// TIA Portal V19 export
FUNCTION_BLOCK "Ventil_Stati"   // FB1095, LAD
TITLE = Ventilstatus
{ S7_Optimized_Access := 'TRUE' }
// 0: geschlossen (grau)
// 1: geöffnet (grün)
// 2: Störung (rot)
// stored: AutoNumber false, MemoryReserve 100, SetENOAutomatically false
   VAR RETAIN
      Param { ExternalAccessible := 'False'; ExternalVisible := 'False'; ExternalWritable := 'False'} : Struct
         "TO" : Time := T#20s;
      END_STRUCT;
      Mld : Struct
         "TO_auf_CM01.QM18" : Bool;
         "TO_zu_CM01.QM18" : Bool;
         "SF_CM01.QM18" : Bool;
         "TO_auf_CM01.QM19" : Bool;
         "TO_zu_CM01.QM19" : Bool;
         "SF_CM01.QM19" : Bool;
         "TO_auf_CM01.QM20" : Bool;
         "TO_zu_CM01.QM20" : Bool;
         "SF_CM01.QM20" : Bool;
         "TO_auf_CM01.QM25" : Bool;
         "TO_zu_CM01.QM25" : Bool;
         "SF_CM01.QM25" : Bool;
         "TO_auf_CM01.QM26" : Bool;
         "TO_zu_CM01.QM26" : Bool;
         "SF_CM01.QM26" : Bool;
         "TO_auf_CM01.QM27" : Bool;
         "TO_zu_CM01.QM27" : Bool;
         "SF_CM01.QM27" : Bool;
         "TO_auf_CM02.QM55" : Bool;
         "TO_zu_CM02.QM55" : Bool;
         "SF_CM02.QM55" : Bool;
         "TO_auf_CM02.QM56" : Bool;
         "TO_zu_CM02.QM56" : Bool;
         "SF_CM02.QM56" : Bool;
         "TO_auf_CM02.QM57" : Bool;
         "TO_zu_CM02.QM57" : Bool;
         "SF_CM02.QM57" : Bool;
         "TO_auf_CM02.QM62" : Bool;
         "TO_zu_CM02.QM62" : Bool;
         "SF_CM02.QM62" : Bool;
         "TO_auf_CM02.QM63" : Bool;
         "TO_zu_CM02.QM63" : Bool;
         "SF_CM02.QM63" : Bool;
         "TO_auf_CM02.QM64" : Bool;
         "TO_zu_CM02.QM64" : Bool;
         "SF_CM02.QM64" : Bool;
         "TO_auf_HQ01.QM21" : Bool;
         "TO_zu_HQ01.QM21" : Bool;
         "SF_HQ01.QM21" : Bool;
         "TO_auf_HQ01.QM22" : Bool;
         "TO_zu_HQ01.QM22" : Bool;
         "SF_HQ01.QM22" : Bool;
         "TO_auf_HQ01.QM23" : Bool;
         "TO_zu_HQ01.QM23" : Bool;
         "SF_HQ01.QM23" : Bool;
         "TO_auf_HQ01.QM24" : Bool;
         "TO_zu_HQ01.QM24" : Bool;
         "SF_HQ01.QM24" : Bool;
         "TO_auf_HQ01.LV01" : Bool;
         "TO_zu_HQ01.LV01" : Bool;
         "SF_HQ01.LV01" : Bool;
         "TO_auf_HQ02.QM58" : Bool;
         "TO_zu_HQ02.QM58" : Bool;
         "SF_HQ02.QM58" : Bool;
         "TO_auf_HQ02.QM59" : Bool;
         "TO_zu_HQ02.QM59" : Bool;
         "SF_HQ02.QM59" : Bool;
         "TO_auf_HQ02.QM60" : Bool;
         "TO_zu_HQ02.QM60" : Bool;
         "SF_HQ02.QM60" : Bool;
         "TO_auf_HQ02.QM61" : Bool;
         "TO_zu_HQ02.QM61" : Bool;
         "SF_HQ02.QM61" : Bool;
         "TO_auf_HQ02.LV02" : Bool;
         "TO_zu_HQ02.LV02" : Bool;
         "SF_HQ02.LV02" : Bool;
         "TO_auf_CM03.QM33" : Bool;
         "TO_zu_CM03.QM33" : Bool;
         "SF_CM03.QM33" : Bool;
         "TO_auf_CM03.QM34" : Bool;
         "TO_zu_CM03.QM34" : Bool;
         "SF_CM03.QM34" : Bool;
         "TO_auf_CM04.QM72" : Bool;
         "TO_zu_CM04.QM72" : Bool;
         "SF_CM04.QM72" : Bool;
         "TO_auf_CM04.QM73" : Bool;
         "TO_zu_CM04.QM73" : Bool;
         "SF_CM04.QM73" : Bool;
         "TO_auf_CM05.QM61" : Bool;
         "TO_zu_CM05.QM61" : Bool;
         "SF_CM05.QM61" : Bool;
         "TO_auf_CM05.QM64" : Bool;
         "TO_zu_CM05.QM64" : Bool;
         "SF_CM05.QM64" : Bool;
         "TO_auf_GP01.QM14" : Bool;
         "TO_zu_GP01.QM14" : Bool;
         "SF_GP01.QM14" : Bool;
         "TO_auf_GP01.QM15" : Bool;
         "TO_zu_GP01.QM15" : Bool;
         "SF_GP01.QM15" : Bool;
         "TO_auf_GP01.QM16" : Bool;
         "TO_zu_GP01.QM16" : Bool;
         "SF_GP01.QM16" : Bool;
         "TO_auf_GP01.QM17" : Bool;
         "TO_zu_GP01.QM17" : Bool;
         "SF_GP01.QM17" : Bool;
         "TO_auf_GP01.QM18" : Bool;
         "TO_zu_GP01.QM18" : Bool;
         "SF_GP01.QM18" : Bool;
         "TO_auf_GP01.QM19" : Bool;
         "TO_zu_GP01.QM19" : Bool;
         "SF_GP01.QM19" : Bool;
         "TO_auf_GP01.QM20" : Bool;
         "TO_zu_GP01.QM20" : Bool;
         "SF_GP01.QM20" : Bool;
         "TO_auf_GP01.QM21" : Bool;
         "TO_zu_GP01.QM21" : Bool;
         "SF_GP01.QM21" : Bool;
         "TO_auf_GP01.QM22" : Bool;
         "TO_zu_GP01.QM22" : Bool;
         "SF_GP01.QM22" : Bool;
         "TO_auf_GP02.QM38" : Bool;
         "TO_zu_GP02.QM38" : Bool;
         "SF_GP02.QM38" : Bool;
         "TO_auf_GP02.QM39" : Bool;
         "TO_zu_GP02.QM39" : Bool;
         "SF_GP02.QM39" : Bool;
         "TO_auf_GP02.QM40" : Bool;
         "TO_zu_GP02.QM40" : Bool;
         "SF_GP02.QM40" : Bool;
         "TO_auf_GP02.QM41" : Bool;
         "TO_zu_GP02.QM41" : Bool;
         "SF_GP02.QM41" : Bool;
         "TO_auf_GP02.QM42" : Bool;
         "TO_zu_GP02.QM42" : Bool;
         "SF_GP02.QM42" : Bool;
         "TO_auf_GP02.QM43" : Bool;
         "TO_zu_GP02.QM43" : Bool;
         "SF_GP02.QM43" : Bool;
         "TO_auf_GP02.QM44" : Bool;
         "TO_zu_GP02.QM44" : Bool;
         "SF_GP02.QM44" : Bool;
         "TO_auf_GP02.QM45" : Bool;
         "TO_zu_GP02.QM45" : Bool;
         "SF_GP02.QM45" : Bool;
         "TO_auf_GP02.QM46" : Bool;
         "TO_zu_GP02.QM46" : Bool;
         "SF_GP02.QM46" : Bool;
      END_STRUCT;
   END_VAR
   VAR
      IEC_Timer { ExternalAccessible := 'False'; ExternalVisible := 'False'; ExternalWritable := 'False'} : Struct
         "TO_auf_CM01.QM18" { S7_SetPoint := 'True'} : TON_TIME;
         "TO_zu_CM01.QM18" { S7_SetPoint := 'True'} : TON_TIME;
         "TO_auf_CM01.QM19" { S7_SetPoint := 'True'} : TON_TIME;
         "TO_zu_CM01.QM19" { S7_SetPoint := 'True'} : TON_TIME;
         "TO_auf_CM01.QM20" { S7_SetPoint := 'True'} : TON_TIME;
         "TO_zu_CM01.QM20" { S7_SetPoint := 'True'} : TON_TIME;
         "TO_auf_CM01.QM25" { S7_SetPoint := 'True'} : TON_TIME;
         "TO_zu_CM01.QM25" { S7_SetPoint := 'True'} : TON_TIME;
         "TO_auf_CM01.QM26" { S7_SetPoint := 'True'} : TON_TIME;
         "TO_zu_CM01.QM26" { S7_SetPoint := 'True'} : TON_TIME;
         "TO_auf_CM01.QM27" { S7_SetPoint := 'True'} : TON_TIME;
         "TO_zu_CM01.QM27" { S7_SetPoint := 'True'} : TON_TIME;
         "TO_auf_CM02.QM55" { S7_SetPoint := 'True'} : TON_TIME;
         "TO_zu_CM02.QM55" { S7_SetPoint := 'True'} : TON_TIME;
         "TO_auf_CM02.QM56" { S7_SetPoint := 'True'} : TON_TIME;
         "TO_zu_CM02.QM56" { S7_SetPoint := 'True'} : TON_TIME;
         "TO_auf_CM02.QM57" { S7_SetPoint := 'True'} : TON_TIME;
         "TO_zu_CM02.QM57" { S7_SetPoint := 'True'} : TON_TIME;
         "TO_auf_CM02.QM62" { S7_SetPoint := 'True'} : TON_TIME;
         "TO_zu_CM02.QM62" { S7_SetPoint := 'True'} : TON_TIME;
         "TO_auf_CM02.QM63" { S7_SetPoint := 'True'} : TON_TIME;
         "TO_zu_CM02.QM63" { S7_SetPoint := 'True'} : TON_TIME;
         "TO_auf_CM02.QM64" { S7_SetPoint := 'True'} : TON_TIME;
         "TO_zu_CM02.QM64" { S7_SetPoint := 'True'} : TON_TIME;
         "TO_auf_HQ01.QM21" { S7_SetPoint := 'True'} : TON_TIME;
         "TO_zu_HQ01.QM21" { S7_SetPoint := 'True'} : TON_TIME;
         "TO_auf_HQ01.QM22" { S7_SetPoint := 'True'} : TON_TIME;
         "TO_zu_HQ01.QM22" { S7_SetPoint := 'True'} : TON_TIME;
         "TO_auf_HQ01.QM23" { S7_SetPoint := 'True'} : TON_TIME;
         "TO_zu_HQ01.QM23" { S7_SetPoint := 'True'} : TON_TIME;
         "TO_auf_HQ01.QM24" { S7_SetPoint := 'True'} : TON_TIME;
         "TO_zu_HQ01.QM24" { S7_SetPoint := 'True'} : TON_TIME;
         "TO_auf_HQ01.LV01" { S7_SetPoint := 'True'} : TON_TIME;
         "TO_zu_HQ01.LV01" { S7_SetPoint := 'True'} : TON_TIME;
         "TO_auf_HQ02.QM58" { S7_SetPoint := 'True'} : TON_TIME;
         "TO_zu_HQ02.QM58" { S7_SetPoint := 'True'} : TON_TIME;
         "TO_auf_HQ02.QM59" { S7_SetPoint := 'True'} : TON_TIME;
         "TO_zu_HQ02.QM59" { S7_SetPoint := 'True'} : TON_TIME;
         "TO_auf_HQ02.QM60" { S7_SetPoint := 'True'} : TON_TIME;
         "TO_zu_HQ02.QM60" { S7_SetPoint := 'True'} : TON_TIME;
         "TO_auf_HQ02.QM61" { S7_SetPoint := 'True'} : TON_TIME;
         "TO_zu_HQ02.QM61" { S7_SetPoint := 'True'} : TON_TIME;
         "TO_auf_HQ02.LV02" { S7_SetPoint := 'True'} : TON_TIME;
         "TO_zu_HQ02.LV02" { S7_SetPoint := 'True'} : TON_TIME;
         "TO_auf_CM03.QM33" { S7_SetPoint := 'True'} : TON_TIME;
         "TO_zu_CM03.QM33" { S7_SetPoint := 'True'} : TON_TIME;
         "TO_auf_CM03.QM34" { S7_SetPoint := 'True'} : TON_TIME;
         "TO_zu_CM03.QM34" { S7_SetPoint := 'True'} : TON_TIME;
         "TO_auf_CM04.QM72" { S7_SetPoint := 'True'} : TON_TIME;
         "TO_zu_CM04.QM72" { S7_SetPoint := 'True'} : TON_TIME;
         "TO_auf_CM04.QM73" { S7_SetPoint := 'True'} : TON_TIME;
         "TO_zu_CM04.QM73" { S7_SetPoint := 'True'} : TON_TIME;
         "TO_auf_CM05.QM61" { S7_SetPoint := 'True'} : TON_TIME;
         "TO_zu_CM05.QM61" { S7_SetPoint := 'True'} : TON_TIME;
         "TO_auf_CM05.QM64" { S7_SetPoint := 'True'} : TON_TIME;
         "TO_zu_CM05.QM64" { S7_SetPoint := 'True'} : TON_TIME;
         "TO_auf_GP01.QM14" { S7_SetPoint := 'True'} : TON_TIME;
         "TO_zu_GP01.QM14" { S7_SetPoint := 'True'} : TON_TIME;
         "TO_auf_GP01.QM15" { S7_SetPoint := 'True'} : TON_TIME;
         "TO_zu_GP01.QM15" { S7_SetPoint := 'True'} : TON_TIME;
         "TO_auf_GP01.QM16" { S7_SetPoint := 'True'} : TON_TIME;
         "TO_zu_GP01.QM16" { S7_SetPoint := 'True'} : TON_TIME;
         "TO_auf_GP01.QM17" { S7_SetPoint := 'True'} : TON_TIME;
         "TO_zu_GP01.QM17" { S7_SetPoint := 'True'} : TON_TIME;
         "TO_auf_GP01.QM18" { S7_SetPoint := 'True'} : TON_TIME;
         "TO_zu_GP01.QM18" { S7_SetPoint := 'True'} : TON_TIME;
         "TO_auf_GP01.QM19" { S7_SetPoint := 'True'} : TON_TIME;
         "TO_zu_GP01.QM19" { S7_SetPoint := 'True'} : TON_TIME;
         "TO_auf_GP01.QM20" { S7_SetPoint := 'True'} : TON_TIME;
         "TO_zu_GP01.QM20" { S7_SetPoint := 'True'} : TON_TIME;
         "TO_auf_GP01.QM21" { S7_SetPoint := 'True'} : TON_TIME;
         "TO_zu_GP01.QM21" { S7_SetPoint := 'True'} : TON_TIME;
         "TO_auf_GP01.QM22" { S7_SetPoint := 'True'} : TON_TIME;
         "TO_zu_GP01.QM22" { S7_SetPoint := 'True'} : TON_TIME;
         "TO_auf_GP02.QM38" { S7_SetPoint := 'True'} : TON_TIME;
         "TO_zu_GP02.QM38" { S7_SetPoint := 'True'} : TON_TIME;
         "TO_auf_GP02.QM39" { S7_SetPoint := 'True'} : TON_TIME;
         "TO_zu_GP02.QM39" { S7_SetPoint := 'True'} : TON_TIME;
         "TO_auf_GP02.QM40" { S7_SetPoint := 'True'} : TON_TIME;
         "TO_zu_GP02.QM40" { S7_SetPoint := 'True'} : TON_TIME;
         "TO_auf_GP02.QM41" { S7_SetPoint := 'True'} : TON_TIME;
         "TO_zu_GP02.QM41" { S7_SetPoint := 'True'} : TON_TIME;
         "TO_auf_GP02.QM42" { S7_SetPoint := 'True'} : TON_TIME;
         "TO_zu_GP02.QM42" { S7_SetPoint := 'True'} : TON_TIME;
         "TO_auf_GP02.QM43" { S7_SetPoint := 'True'} : TON_TIME;
         "TO_zu_GP02.QM43" { S7_SetPoint := 'True'} : TON_TIME;
         "TO_auf_GP02.QM44" { S7_SetPoint := 'True'} : TON_TIME;
         "TO_zu_GP02.QM44" { S7_SetPoint := 'True'} : TON_TIME;
         "TO_auf_GP02.QM45" { S7_SetPoint := 'True'} : TON_TIME;
         "TO_zu_GP02.QM45" { S7_SetPoint := 'True'} : TON_TIME;
         "TO_auf_GP02.QM46" { S7_SetPoint := 'True'} : TON_TIME;
         "TO_zu_GP02.QM46" { S7_SetPoint := 'True'} : TON_TIME;
      END_STRUCT;
   END_VAR
   VAR CONSTANT
      grau : USInt;
      grün : USInt := 1;
      rot : USInt := 2;
   END_VAR
BEGIN

REGION Network 1 (SCL): CM01

   "Ventilstatus"(SRM_auf:= "E_SRM_CM01.QM18_auf",
                  SRM_zu:= "E_SRM_CM01.QM18_zu",
                  A_Ventil:= "A_CM01.QM18",
                  Zeit:= #Param.TO,
                  "Farbe HMI"=> "Panel".Ventil."CM01.QM18",
                  Mld_Sensorfehler:= #Mld."SF_CM01.QM18",
                  Mld_TO_oeffnen=> #Mld."TO_auf_CM01.QM18",
                  Mld_TO_schliessen=> #Mld."TO_zu_CM01.QM18",
                  TO_oeffnen:= #IEC_Timer."TO_auf_CM01.QM18",
                  TO_schliessen:= #IEC_Timer."TO_zu_CM01.QM18");

   "Ventilstatus"(SRM_auf := "E_SRM_CM01.QM19_auf",
                  SRM_zu := "E_SRM_CM01.QM19_zu",
                  A_Ventil := "A_CM01.QM19",
                  Zeit := #Param.TO,
                  "Farbe HMI" => "Panel".Ventil."CM01.QM19",
                  Mld_Sensorfehler := #Mld."SF_CM01.QM19",
                  Mld_TO_oeffnen => #Mld."TO_auf_CM01.QM19",
                  Mld_TO_schliessen => #Mld."TO_zu_CM01.QM19",
                  TO_oeffnen := #IEC_Timer."TO_auf_CM01.QM19",
                  TO_schliessen := #IEC_Timer."TO_zu_CM01.QM19");

   "Ventilstatus"(SRM_auf := "E_SRM_CM01.QM20_auf",
                  SRM_zu := "E_SRM_CM01.QM20_zu",
                  A_Ventil := "A_CM01.QM20",
                  Zeit := #Param.TO,
                  "Farbe HMI" => "Panel".Ventil."CM01.QM20",
                  Mld_Sensorfehler := #Mld."SF_CM01.QM20",
                  Mld_TO_oeffnen => #Mld."TO_auf_CM01.QM20",
                  Mld_TO_schliessen => #Mld."TO_zu_CM01.QM20",
                  TO_oeffnen := #IEC_Timer."TO_auf_CM01.QM20",
                  TO_schliessen := #IEC_Timer."TO_zu_CM01.QM20");

   "Ventilstatus"(SRM_auf := "E_SRM_CM01.QM25_auf",
                  SRM_zu := "E_SRM_CM01.QM25_zu",
                  A_Ventil := "A_CM01.QM25",
                  Zeit := #Param.TO,
                  "Farbe HMI" => "Panel".Ventil."CM01.QM25",
                  Mld_Sensorfehler := #Mld."SF_CM01.QM25",
                  Mld_TO_oeffnen => #Mld."TO_auf_CM01.QM25",
                  Mld_TO_schliessen => #Mld."TO_zu_CM01.QM25",
                  TO_oeffnen := #IEC_Timer."TO_auf_CM01.QM25",
                  TO_schliessen := #IEC_Timer."TO_zu_CM01.QM25");

   "Ventilstatus"(SRM_auf := "E_SRM_CM01.QM26_auf",
                  SRM_zu := "E_SRM_CM01.QM26_zu",
                  A_Ventil := "A_CM01.QM26",
                  Zeit := #Param.TO,
                  "Farbe HMI" => "Panel".Ventil."CM01.QM26",
                  Mld_Sensorfehler := #Mld."SF_CM01.QM26",
                  Mld_TO_oeffnen => #Mld."TO_auf_CM01.QM26",
                  Mld_TO_schliessen => #Mld."TO_zu_CM01.QM26",
                  TO_oeffnen := #IEC_Timer."TO_auf_CM01.QM26",
                  TO_schliessen := #IEC_Timer."TO_zu_CM01.QM26");

   "Ventilstatus"(SRM_auf := "E_SRM_CM01.QM27_auf",
                  SRM_zu := "E_SRM_CM01.QM27_zu",
                  A_Ventil := "A_CM01.QM27",
                  Zeit := #Param.TO,
                  "Farbe HMI" => "Panel".Ventil."CM01.QM27",
                  Mld_Sensorfehler := #Mld."SF_CM01.QM27",
                  Mld_TO_oeffnen => #Mld."TO_auf_CM01.QM27",
                  Mld_TO_schliessen => #Mld."TO_zu_CM01.QM27",
                  TO_oeffnen := #IEC_Timer."TO_auf_CM01.QM27",
                  TO_schliessen := #IEC_Timer."TO_zu_CM01.QM27");
END_REGION

REGION Network 2 (SCL): HQ01
   "Ventilstatus"(SRM_auf := "E_SRM_HQ01.LV01_auf",
                  SRM_zu := "E_SRM_HQ01.LV01_zu",
                  A_Ventil := "A_HQ01.LV01",
                  Zeit := #Param.TO,
                  "Farbe HMI" => "Panel".Ventil."HQ01.LV01",
                  Mld_Sensorfehler := #Mld."SF_HQ01.LV01",
                  Mld_TO_oeffnen => #Mld."TO_auf_HQ01.LV01",
                  Mld_TO_schliessen => #Mld."TO_zu_HQ01.LV01",
                  TO_oeffnen := #IEC_Timer."TO_auf_HQ01.LV01",
                  TO_schliessen := #IEC_Timer."TO_zu_HQ01.LV01");

   "Ventilstatus"(SRM_auf := "E_SRM_HQ01.QM21_auf",
                  SRM_zu := "E_SRM_HQ01.QM21_zu",
                  A_Ventil := "A_HQ01.QM21",
                  Zeit := #Param.TO,
                  "Farbe HMI" => "Panel".Ventil."HQ01.QM21",
                  Mld_Sensorfehler := #Mld."SF_HQ01.QM21",
                  Mld_TO_oeffnen => #Mld."TO_auf_HQ01.QM21",
                  Mld_TO_schliessen => #Mld."TO_zu_HQ01.QM21",
                  TO_oeffnen := #IEC_Timer."TO_auf_HQ01.QM21",
                  TO_schliessen := #IEC_Timer."TO_zu_HQ01.QM21");

   "Ventilstatus"(SRM_auf := "E_SRM_HQ01.QM22_auf",
                  SRM_zu := "E_SRM_HQ01.QM22_zu",
                  A_Ventil := "A_HQ01.QM22",
                  Zeit := #Param.TO,
                  "Farbe HMI" => "Panel".Ventil."HQ01.QM22",
                  Mld_Sensorfehler := #Mld."SF_HQ01.QM22",
                  Mld_TO_oeffnen => #Mld."TO_auf_HQ01.QM22",
                  Mld_TO_schliessen => #Mld."TO_zu_HQ01.QM22",
                  TO_oeffnen := #IEC_Timer."TO_auf_HQ01.QM22",
                  TO_schliessen := #IEC_Timer."TO_zu_HQ01.QM22");

   "Ventilstatus"(SRM_auf := "E_SRM_HQ01.QM23_auf",
                  SRM_zu := "E_SRM_HQ01.QM23_zu",
                  A_Ventil := "A_HQ01.QM23",
                  Zeit := #Param.TO,
                  "Farbe HMI" => "Panel".Ventil."HQ01.QM23",
                  Mld_Sensorfehler := #Mld."SF_HQ01.QM23",
                  Mld_TO_oeffnen => #Mld."TO_auf_HQ01.QM23",
                  Mld_TO_schliessen => #Mld."TO_zu_HQ01.QM23",
                  TO_oeffnen := #IEC_Timer."TO_auf_HQ01.QM23",
                  TO_schliessen := #IEC_Timer."TO_zu_HQ01.QM23");

   "Ventilstatus"(SRM_auf := "E_SRM_HQ01.QM24_auf",
                  SRM_zu := "E_SRM_HQ01.QM24_zu",
                  A_Ventil := "A_HQ01.QM24",
                  Zeit := #Param.TO,
                  "Farbe HMI" => "Panel".Ventil."HQ01.QM24",
                  Mld_Sensorfehler := #Mld."SF_HQ01.QM24",
                  Mld_TO_oeffnen => #Mld."TO_auf_HQ01.QM24",
                  Mld_TO_schliessen => #Mld."TO_zu_HQ01.QM24",
                  TO_oeffnen := #IEC_Timer."TO_auf_HQ01.QM24",
                  TO_schliessen := #IEC_Timer."TO_zu_HQ01.QM24");
END_REGION

REGION Network 3 (SCL): CM03

   "Ventilstatus"(SRM_auf := "E_SRM_CM03.QM33_auf",
                  SRM_zu := "E_SRM_CM03.QM33_zu",
                  A_Ventil := "A_CM03.QM33",
                  Zeit := #Param.TO,
                  "Farbe HMI" => "Panel".Ventil."CM03.QM33",
                  Mld_Sensorfehler := #Mld."SF_CM03.QM33",
                  Mld_TO_oeffnen => #Mld."TO_auf_CM03.QM33",
                  Mld_TO_schliessen => #Mld."TO_zu_CM03.QM33",
                  TO_oeffnen := #IEC_Timer."TO_auf_CM03.QM33",
                  TO_schliessen := #IEC_Timer."TO_zu_CM03.QM33");

   "Ventilstatus"(SRM_auf := "E_SRM_CM03.QM34_auf",
                  SRM_zu := "E_SRM_CM03.QM34_zu",
                  A_Ventil := "A_CM03.QM34",
                  Zeit := #Param.TO,
                  "Farbe HMI" => "Panel".Ventil."CM03.QM34",
                  Mld_Sensorfehler := #Mld."SF_CM03.QM34",
                  Mld_TO_oeffnen => #Mld."TO_auf_CM03.QM34",
                  Mld_TO_schliessen => #Mld."TO_zu_CM03.QM34",
                  TO_oeffnen := #IEC_Timer."TO_auf_CM03.QM34",
                  TO_schliessen := #IEC_Timer."TO_zu_CM03.QM34");

   "Ventilstatus_einfach"(A_Ventil:="A_CM03.QM35",
                          "Farbe HMI"=>"Panel".Ventil."CM03.QM35");

   "Ventilstatus_einfach"(A_Ventil := "A_CM03.QM36",
                          "Farbe HMI" => "Panel".Ventil."CM03.QM36");

   "Ventilstatus_einfach"(A_Ventil := "A_CM03.QM37",
                          "Farbe HMI" => "Panel".Ventil."CM03.QM37");
END_REGION

REGION Network 4 (SCL): CM02

   "Ventilstatus"(SRM_auf := "E_SRM_CM02.QM55_auf",
                  SRM_zu := "E_SRM_CM02.QM55_zu",
                  A_Ventil := "A_CM02.QM55",
                  Zeit := #Param.TO,
                  "Farbe HMI" => "Panel".Ventil."CM02.QM55",
                  Mld_Sensorfehler := #Mld."SF_CM02.QM55",
                  Mld_TO_oeffnen => #Mld."TO_auf_CM02.QM55",
                  Mld_TO_schliessen => #Mld."TO_zu_CM02.QM55",
                  TO_oeffnen := #IEC_Timer."TO_auf_CM02.QM55",
                  TO_schliessen := #IEC_Timer."TO_zu_CM02.QM55");

   "Ventilstatus"(SRM_auf := "E_SRM_CM02.QM56_auf",
                  SRM_zu := "E_SRM_CM02.QM56_zu",
                  A_Ventil := "A_CM02.QM56",
                  Zeit := #Param.TO,
                  "Farbe HMI" => "Panel".Ventil."CM02.QM56",
                  Mld_Sensorfehler := #Mld."SF_CM02.QM56",
                  Mld_TO_oeffnen => #Mld."TO_auf_CM02.QM56",
                  Mld_TO_schliessen => #Mld."TO_zu_CM02.QM56",
                  TO_oeffnen := #IEC_Timer."TO_auf_CM02.QM56",
                  TO_schliessen := #IEC_Timer."TO_zu_CM02.QM56");

   "Ventilstatus"(SRM_auf := "E_SRM_CM02.QM57_auf",
                  SRM_zu := "E_SRM_CM02.QM57_zu",
                  A_Ventil := "A_CM02.QM57",
                  Zeit := #Param.TO,
                  "Farbe HMI" => "Panel".Ventil."CM02.QM57",
                  Mld_Sensorfehler := #Mld."SF_CM02.QM57",
                  Mld_TO_oeffnen => #Mld."TO_auf_CM02.QM57",
                  Mld_TO_schliessen => #Mld."TO_zu_CM02.QM57",
                  TO_oeffnen := #IEC_Timer."TO_auf_CM02.QM57",
                  TO_schliessen := #IEC_Timer."TO_zu_CM02.QM57");

   "Ventilstatus"(SRM_auf := "E_SRM_CM02.QM62_auf",
                  SRM_zu := "E_SRM_CM02.QM62_zu",
                  A_Ventil := "A_CM02.QM62",
                  Zeit := #Param.TO,
                  "Farbe HMI" => "Panel".Ventil."CM02.QM62",
                  Mld_Sensorfehler := #Mld."SF_CM02.QM62",
                  Mld_TO_oeffnen => #Mld."TO_auf_CM02.QM62",
                  Mld_TO_schliessen => #Mld."TO_zu_CM02.QM62",
                  TO_oeffnen := #IEC_Timer."TO_auf_CM02.QM62",
                  TO_schliessen := #IEC_Timer."TO_zu_CM02.QM62");

   "Ventilstatus"(SRM_auf := "E_SRM_CM02.QM63_auf",
                  SRM_zu := "E_SRM_CM02.QM63_zu",
                  A_Ventil := "A_CM02.QM63",
                  Zeit := #Param.TO,
                  "Farbe HMI" => "Panel".Ventil."CM02.QM63",
                  Mld_Sensorfehler := #Mld."SF_CM02.QM63",
                  Mld_TO_oeffnen => #Mld."TO_auf_CM02.QM63",
                  Mld_TO_schliessen => #Mld."TO_zu_CM02.QM63",
                  TO_oeffnen := #IEC_Timer."TO_auf_CM02.QM63",
                  TO_schliessen := #IEC_Timer."TO_zu_CM02.QM63");

   "Ventilstatus"(SRM_auf := "E_SRM_CM02.QM64_auf",
                  SRM_zu := "E_SRM_CM02.QM64_zu",
                  A_Ventil := "A_CM02.QM64",
                  Zeit := #Param.TO,
                  "Farbe HMI" => "Panel".Ventil."CM02.QM64",
                  Mld_Sensorfehler := #Mld."SF_CM02.QM64",
                  Mld_TO_oeffnen => #Mld."TO_auf_CM02.QM64",
                  Mld_TO_schliessen => #Mld."TO_zu_CM02.QM64",
                  TO_oeffnen := #IEC_Timer."TO_auf_CM02.QM64",
                  TO_schliessen := #IEC_Timer."TO_zu_CM02.QM64");
END_REGION

REGION Network 5 (SCL): HQ02
   "Ventilstatus"(SRM_auf := "E_SRM_HQ02.LV02_auf",
                  SRM_zu := "E_SRM_HQ02.LV02_zu",
                  A_Ventil := "A_HQ02.LV02",
                  Zeit := #Param.TO,
                  "Farbe HMI" => "Panel".Ventil."HQ02.LV02",
                  Mld_Sensorfehler := #Mld."SF_HQ02.LV02",
                  Mld_TO_oeffnen => #Mld."TO_auf_HQ02.LV02",
                  Mld_TO_schliessen => #Mld."TO_zu_HQ02.LV02",
                  TO_oeffnen := #IEC_Timer."TO_auf_HQ02.LV02",
                  TO_schliessen := #IEC_Timer."TO_zu_HQ02.LV02");

   "Ventilstatus"(SRM_auf := "E_SRM_HQ02.QM58_auf",
                  SRM_zu := "E_SRM_HQ02.QM58_zu",
                  A_Ventil := "A_HQ02.QM58",
                  Zeit := #Param.TO,
                  "Farbe HMI" => "Panel".Ventil."HQ02.QM58",
                  Mld_Sensorfehler := #Mld."SF_HQ02.QM58",
                  Mld_TO_oeffnen => #Mld."TO_auf_HQ02.QM58",
                  Mld_TO_schliessen => #Mld."TO_zu_HQ02.QM58",
                  TO_oeffnen := #IEC_Timer."TO_auf_HQ02.QM58",
                  TO_schliessen := #IEC_Timer."TO_zu_HQ02.QM58");

   "Ventilstatus"(SRM_auf := "E_SRM_HQ02.QM59_auf",
                  SRM_zu := "E_SRM_HQ02.QM59_zu",
                  A_Ventil := "A_HQ02.QM59",
                  Zeit := #Param.TO,
                  "Farbe HMI" => "Panel".Ventil."HQ02.QM59",
                  Mld_Sensorfehler := #Mld."SF_HQ02.QM59",
                  Mld_TO_oeffnen => #Mld."TO_auf_HQ02.QM59",
                  Mld_TO_schliessen => #Mld."TO_zu_HQ02.QM59",
                  TO_oeffnen := #IEC_Timer."TO_auf_HQ02.QM59",
                  TO_schliessen := #IEC_Timer."TO_zu_HQ02.QM59");

   "Ventilstatus"(SRM_auf := "E_SRM_HQ02.QM60_auf",
                  SRM_zu := "E_SRM_HQ02.QM60_zu",
                  A_Ventil := "A_HQ02.QM60",
                  Zeit := #Param.TO,
                  "Farbe HMI" => "Panel".Ventil."HQ02.QM60",
                  Mld_Sensorfehler := #Mld."SF_HQ02.QM60",
                  Mld_TO_oeffnen => #Mld."TO_auf_HQ02.QM60",
                  Mld_TO_schliessen => #Mld."TO_zu_HQ02.QM60",
                  TO_oeffnen := #IEC_Timer."TO_auf_HQ02.QM60",
                  TO_schliessen := #IEC_Timer."TO_zu_HQ02.QM60");

   "Ventilstatus"(SRM_auf := "E_SRM_HQ02.QM61_auf",
                  SRM_zu := "E_SRM_HQ02.QM61_zu",
                  A_Ventil := "A_HQ02.QM61",
                  Zeit := #Param.TO,
                  "Farbe HMI" => "Panel".Ventil."HQ02.QM61",
                  Mld_Sensorfehler := #Mld."SF_HQ02.QM61",
                  Mld_TO_oeffnen => #Mld."TO_auf_HQ02.QM61",
                  Mld_TO_schliessen => #Mld."TO_zu_HQ02.QM61",
                  TO_oeffnen := #IEC_Timer."TO_auf_HQ02.QM61",
                  TO_schliessen := #IEC_Timer."TO_zu_HQ02.QM61");
END_REGION

REGION Network 6 (SCL): CM04

   "Ventilstatus"(SRM_auf := "E_SRM_CM04.QM72_auf",
                  SRM_zu := "E_SRM_CM04.QM72_zu",
                  A_Ventil := "A_CM04.QM72",
                  Zeit := #Param.TO,
                  "Farbe HMI" => "Panel".Ventil."CM04.QM72",
                  Mld_Sensorfehler := #Mld."SF_CM04.QM72",
                  Mld_TO_oeffnen => #Mld."TO_auf_CM04.QM72",
                  Mld_TO_schliessen => #Mld."TO_zu_CM04.QM72",
                  TO_oeffnen := #IEC_Timer."TO_auf_CM04.QM72",
                  TO_schliessen := #IEC_Timer."TO_zu_CM04.QM72");

   "Ventilstatus"(SRM_auf := "E_SRM_CM04.QM73_auf",
                  SRM_zu := "E_SRM_CM04.QM73_zu",
                  A_Ventil := "A_CM04.QM73",
                  Zeit := #Param.TO,
                  "Farbe HMI" => "Panel".Ventil."CM04.QM73",
                  Mld_Sensorfehler := #Mld."SF_CM04.QM73",
                  Mld_TO_oeffnen => #Mld."TO_auf_CM04.QM73",
                  Mld_TO_schliessen => #Mld."TO_zu_CM04.QM73",
                  TO_oeffnen := #IEC_Timer."TO_auf_CM04.QM73",
                  TO_schliessen := #IEC_Timer."TO_zu_CM04.QM73");

   "Ventilstatus_einfach"(A_Ventil := "A_CM04.QM74",
                          "Farbe HMI" => "Panel".Ventil."CM04.QM74");

   "Ventilstatus_einfach"(A_Ventil := "A_CM04.QM75",
                          "Farbe HMI" => "Panel".Ventil."CM04.QM75");

   "Ventilstatus_einfach"(A_Ventil := "A_CM04.QM76",
                          "Farbe HMI" => "Panel".Ventil."CM04.QM76");

   "Ventilstatus_einfach"(A_Ventil := "A_CM04.QM77",
                          "Farbe HMI" => "Panel".Ventil."CM04.QM77");
END_REGION

REGION Network 7 (SCL): CM05
   "Ventilstatus"(SRM_auf := "E_SRM_CM05.QM61_auf",
                  SRM_zu := "E_SRM_CM05.QM61_zu",
                  A_Ventil := "A_CM05.QM61",
                  Zeit := #Param.TO,
                  "Farbe HMI" => "Panel".Ventil."CM05.QM61",
                  Mld_Sensorfehler := #Mld."SF_CM05.QM61",
                  Mld_TO_oeffnen => #Mld."TO_auf_CM05.QM61",
                  Mld_TO_schliessen => #Mld."TO_zu_CM05.QM61",
                  TO_oeffnen := #IEC_Timer."TO_auf_CM05.QM61",
                  TO_schliessen := #IEC_Timer."TO_zu_CM05.QM61");

   "Ventilstatus_einfach"(A_Ventil := "A_CM05.QM62",
                          "Farbe HMI" => "Panel".Ventil."CM05.QM62");

   "Ventilstatus_einfach"(A_Ventil := "A_CM05.QM63",
                          "Farbe HMI" => "Panel".Ventil."CM05.QM63");

   "Ventilstatus"(SRM_auf := "E_SRM_CM05.QM64_auf",
                  SRM_zu := "E_SRM_CM05.QM64_zu",
                  A_Ventil := "A_CM05.QM64",
                  Zeit := #Param.TO,
                  "Farbe HMI" => "Panel".Ventil."CM05.QM64",
                  Mld_Sensorfehler := #Mld."SF_CM05.QM64",
                  Mld_TO_oeffnen => #Mld."TO_auf_CM05.QM64",
                  Mld_TO_schliessen => #Mld."TO_zu_CM05.QM64",
                  TO_oeffnen := #IEC_Timer."TO_auf_CM05.QM64",
                  TO_schliessen := #IEC_Timer."TO_zu_CM05.QM64");
END_REGION

REGION Network 8 (SCL): GP01

   "Ventilstatus"(SRM_auf := "E_SRM_GP01.QM14_auf",
                  SRM_zu := "E_SRM_GP01.QM14_zu",
                  A_Ventil := "A_GP01.QM14",
                  Zeit := #Param.TO,
                  "Farbe HMI" => "Panel".Ventil."GP01.QM14",
                  Mld_Sensorfehler := #Mld."SF_GP01.QM14",
                  Mld_TO_oeffnen => #Mld."TO_auf_GP01.QM14",
                  Mld_TO_schliessen => #Mld."TO_zu_GP01.QM14",
                  TO_oeffnen := #IEC_Timer."TO_auf_GP01.QM14",
                  TO_schliessen := #IEC_Timer."TO_zu_GP01.QM14");

   "Ventilstatus"(SRM_auf := "E_SRM_GP01.QM15_auf",
                  SRM_zu := "E_SRM_GP01.QM15_zu",
                  A_Ventil := "A_GP01.QM15",
                  Zeit := #Param.TO,
                  "Farbe HMI" => "Panel".Ventil."GP01.QM15",
                  Mld_Sensorfehler := #Mld."SF_GP01.QM15",
                  Mld_TO_oeffnen => #Mld."TO_auf_GP01.QM15",
                  Mld_TO_schliessen => #Mld."TO_zu_GP01.QM15",
                  TO_oeffnen := #IEC_Timer."TO_auf_GP01.QM15",
                  TO_schliessen := #IEC_Timer."TO_zu_GP01.QM15");

   "Ventilstatus"(SRM_auf := "E_SRM_GP01.QM16_auf",
                  SRM_zu := "E_SRM_GP01.QM16_zu",
                  A_Ventil := "A_GP01.QM16",
                  Zeit := #Param.TO,
                  "Farbe HMI" => "Panel".Ventil."GP01.QM16",
                  Mld_Sensorfehler := #Mld."SF_GP01.QM16",
                  Mld_TO_oeffnen => #Mld."TO_auf_GP01.QM16",
                  Mld_TO_schliessen => #Mld."TO_zu_GP01.QM16",
                  TO_oeffnen := #IEC_Timer."TO_auf_GP01.QM16",
                  TO_schliessen := #IEC_Timer."TO_zu_GP01.QM16");

   "Ventilstatus"(SRM_auf := "E_SRM_GP01.QM17_auf",
                  SRM_zu := "E_SRM_GP01.QM17_zu",
                  A_Ventil := "A_GP01.QM17",
                  Zeit := #Param.TO,
                  "Farbe HMI" => "Panel".Ventil."GP01.QM17",
                  Mld_Sensorfehler := #Mld."SF_GP01.QM17",
                  Mld_TO_oeffnen => #Mld."TO_auf_GP01.QM17",
                  Mld_TO_schliessen => #Mld."TO_zu_GP01.QM17",
                  TO_oeffnen := #IEC_Timer."TO_auf_GP01.QM17",
                  TO_schliessen := #IEC_Timer."TO_zu_GP01.QM17");

   "Ventilstatus"(SRM_auf := "E_SRM_GP01.QM18_auf",
                  SRM_zu := "E_SRM_GP01.QM18_zu",
                  A_Ventil := "A_GP01.QM18",
                  Zeit := #Param.TO,
                  "Farbe HMI" => "Panel".Ventil."GP01.QM18",
                  Mld_Sensorfehler := #Mld."SF_GP01.QM18",
                  Mld_TO_oeffnen => #Mld."TO_auf_GP01.QM18",
                  Mld_TO_schliessen => #Mld."TO_zu_GP01.QM18",
                  TO_oeffnen := #IEC_Timer."TO_auf_GP01.QM18",
                  TO_schliessen := #IEC_Timer."TO_zu_GP01.QM18");

   "Ventilstatus"(SRM_auf := "E_SRM_GP01.QM19_auf",
                  SRM_zu := "E_SRM_GP01.QM19_zu",
                  A_Ventil := "A_GP01.QM19",
                  Zeit := #Param.TO,
                  "Farbe HMI" => "Panel".Ventil."GP01.QM19",
                  Mld_Sensorfehler := #Mld."SF_GP01.QM19",
                  Mld_TO_oeffnen => #Mld."TO_auf_GP01.QM19",
                  Mld_TO_schliessen => #Mld."TO_zu_GP01.QM19",
                  TO_oeffnen := #IEC_Timer."TO_auf_GP01.QM19",
                  TO_schliessen := #IEC_Timer."TO_zu_GP01.QM19");

   "Ventilstatus"(SRM_auf := "E_SRM_GP01.QM20_auf",
                  SRM_zu := "E_SRM_GP01.QM20_zu",
                  A_Ventil := "A_GP01.QM20",
                  Zeit := #Param.TO,
                  "Farbe HMI" => "Panel".Ventil."GP01.QM20",
                  Mld_Sensorfehler := #Mld."SF_GP01.QM20",
                  Mld_TO_oeffnen => #Mld."TO_auf_GP01.QM20",
                  Mld_TO_schliessen => #Mld."TO_zu_GP01.QM20",
                  TO_oeffnen := #IEC_Timer."TO_auf_GP01.QM20",
                  TO_schliessen := #IEC_Timer."TO_zu_GP01.QM20");

   "Ventilstatus"(SRM_auf := "E_SRM_GP01.QM21_auf",
                  SRM_zu := "E_SRM_GP01.QM21_zu",
                  A_Ventil := "A_GP01.QM21",
                  Zeit := #Param.TO,
                  "Farbe HMI" => "Panel".Ventil."GP01.QM21",
                  Mld_Sensorfehler := #Mld."SF_GP01.QM21",
                  Mld_TO_oeffnen => #Mld."TO_auf_GP01.QM21",
                  Mld_TO_schliessen => #Mld."TO_zu_GP01.QM21",
                  TO_oeffnen := #IEC_Timer."TO_auf_GP01.QM21",
                  TO_schliessen := #IEC_Timer."TO_zu_GP01.QM21");

   "Ventilstatus"(SRM_auf := "E_SRM_GP01.QM22_auf",
                  SRM_zu := "E_SRM_GP01.QM22_zu",
                  A_Ventil := "A_GP01.QM22",
                  Zeit := #Param.TO,
                  "Farbe HMI" => "Panel".Ventil."GP01.QM22",
                  Mld_Sensorfehler := #Mld."SF_GP01.QM22",
                  Mld_TO_oeffnen => #Mld."TO_auf_GP01.QM22",
                  Mld_TO_schliessen => #Mld."TO_zu_GP01.QM22",
                  TO_oeffnen := #IEC_Timer."TO_auf_GP01.QM22",
                  TO_schliessen := #IEC_Timer."TO_zu_GP01.QM22");

   "Ventilstatus_einfach"(A_Ventil:="A_GP01.QM23",
                          "Farbe HMI"=> "Panel".Ventil."GP01.QM23");
END_REGION

REGION Network 9 (SCL): GP02
   "Ventilstatus_einfach"(A_Ventil := "A_GP02.QM37",
                          "Farbe HMI" => "Panel".Ventil."GP02.QM37");

   "Ventilstatus"(SRM_auf := "E_SRM_GP02.QM38_auf",
                  SRM_zu := "E_SRM_GP02.QM38_zu",
                  A_Ventil := "A_GP02.QM38",
                  Zeit := #Param.TO,
                  "Farbe HMI" => "Panel".Ventil."GP02.QM38",
                  Mld_Sensorfehler := #Mld."SF_GP02.QM38",
                  Mld_TO_oeffnen => #Mld."TO_auf_GP02.QM38",
                  Mld_TO_schliessen => #Mld."TO_zu_GP02.QM38",
                  TO_oeffnen := #IEC_Timer."TO_auf_GP02.QM38",
                  TO_schliessen := #IEC_Timer."TO_zu_GP02.QM38");

   "Ventilstatus"(SRM_auf := "E_SRM_GP02.QM39_auf",
                  SRM_zu := "E_SRM_GP02.QM39_zu",
                  A_Ventil := "A_GP02.QM39",
                  Zeit := #Param.TO,
                  "Farbe HMI" => "Panel".Ventil."GP02.QM39",
                  Mld_Sensorfehler := #Mld."SF_GP02.QM39",
                  Mld_TO_oeffnen => #Mld."TO_auf_GP02.QM39",
                  Mld_TO_schliessen => #Mld."TO_zu_GP02.QM39",
                  TO_oeffnen := #IEC_Timer."TO_auf_GP02.QM39",
                  TO_schliessen := #IEC_Timer."TO_zu_GP02.QM39");

   "Ventilstatus"(SRM_auf := "E_SRM_GP02.QM40_auf",
                  SRM_zu := "E_SRM_GP02.QM40_zu",
                  A_Ventil := "A_GP02.QM40",
                  Zeit := #Param.TO,
                  "Farbe HMI" => "Panel".Ventil."GP02.QM40",
                  Mld_Sensorfehler := #Mld."SF_GP02.QM40",
                  Mld_TO_oeffnen => #Mld."TO_auf_GP02.QM40",
                  Mld_TO_schliessen => #Mld."TO_zu_GP02.QM40",
                  TO_oeffnen := #IEC_Timer."TO_auf_GP02.QM40",
                  TO_schliessen := #IEC_Timer."TO_zu_GP02.QM40");

   "Ventilstatus"(SRM_auf := "E_SRM_GP02.QM41_auf",
                  SRM_zu := "E_SRM_GP02.QM41_zu",
                  A_Ventil := "A_GP02.QM41",
                  Zeit := #Param.TO,
                  "Farbe HMI" => "Panel".Ventil."GP02.QM41",
                  Mld_Sensorfehler := #Mld."SF_GP02.QM41",
                  Mld_TO_oeffnen => #Mld."TO_auf_GP02.QM41",
                  Mld_TO_schliessen => #Mld."TO_zu_GP02.QM41",
                  TO_oeffnen := #IEC_Timer."TO_auf_GP02.QM41",
                  TO_schliessen := #IEC_Timer."TO_zu_GP02.QM41");

   "Ventilstatus"(SRM_auf := "E_SRM_GP02.QM42_auf",
                  SRM_zu := "E_SRM_GP02.QM42_zu",
                  A_Ventil := "A_GP02.QM42",
                  Zeit := #Param.TO,
                  "Farbe HMI" => "Panel".Ventil."GP02.QM42",
                  Mld_Sensorfehler := #Mld."SF_GP02.QM42",
                  Mld_TO_oeffnen => #Mld."TO_auf_GP02.QM42",
                  Mld_TO_schliessen => #Mld."TO_zu_GP02.QM41",
                  TO_oeffnen := #IEC_Timer."TO_auf_GP02.QM42",
                  TO_schliessen := #IEC_Timer."TO_zu_GP02.QM42");

   "Ventilstatus"(SRM_auf := "DB_PNOZ_IN_Out".In."SRM_Auf_BG-QM43",
                  SRM_zu := "DB_PNOZ_IN_Out".In."SRM_Zu_BG-QM43",
                  A_Ventil := "A_GP02.QM43",
                  Zeit := #Param.TO,
                  "Farbe HMI" => "Panel".Ventil."GP02.QM43",
                  Mld_Sensorfehler := #Mld."SF_GP02.QM43",
                  Mld_TO_oeffnen => #Mld."TO_auf_GP02.QM43",
                  Mld_TO_schliessen => #Mld."TO_zu_GP02.QM43",
                  TO_oeffnen := #IEC_Timer."TO_auf_GP02.QM43",
                  TO_schliessen := #IEC_Timer."TO_zu_GP02.QM43");

   "Ventilstatus"(SRM_auf := "DB_PNOZ_IN_Out".In."SRM_Auf_BG-QM44",
                  SRM_zu := "DB_PNOZ_IN_Out".In."SRM_Zu_BG-QM44",
                  A_Ventil := "A_GP02.QM44",
                  Zeit := #Param.TO,
                  "Farbe HMI" => "Panel".Ventil."GP02.QM44",
                  Mld_Sensorfehler := #Mld."SF_GP02.QM44",
                  Mld_TO_oeffnen => #Mld."TO_auf_GP02.QM44",
                  Mld_TO_schliessen => #Mld."TO_zu_GP02.QM44",
                  TO_oeffnen := #IEC_Timer."TO_auf_GP02.QM44",
                  TO_schliessen := #IEC_Timer."TO_zu_GP02.QM44");

   "Ventilstatus"(SRM_auf := "E_SRM_GP02.QM45_auf",
                  SRM_zu := "E_SRM_GP02.QM45_zu",
                  A_Ventil := "A_GP02.QM45",
                  Zeit := #Param.TO,
                  "Farbe HMI" => "Panel".Ventil."GP02.QM45",
                  Mld_Sensorfehler := #Mld."SF_GP02.QM45",
                  Mld_TO_oeffnen => #Mld."TO_auf_GP02.QM45",
                  Mld_TO_schliessen => #Mld."TO_zu_GP02.QM45",
                  TO_oeffnen := #IEC_Timer."TO_auf_GP02.QM45",
                  TO_schliessen := #IEC_Timer."TO_zu_GP02.QM45");

   "Ventilstatus"(SRM_auf := "E_SRM_GP02.QM46_auf",
                  SRM_zu := "E_SRM_GP02.QM46_zu",
                  A_Ventil := "A_GP02.QM46",
                  Zeit := #Param.TO,
                  "Farbe HMI" => "Panel".Ventil."GP02.QM46",
                  Mld_Sensorfehler := #Mld."SF_GP02.QM46",
                  Mld_TO_oeffnen => #Mld."TO_auf_GP02.QM46",
                  Mld_TO_schliessen => #Mld."TO_zu_GP02.QM46",
                  TO_oeffnen := #IEC_Timer."TO_auf_GP02.QM46",
                  TO_schliessen := #IEC_Timer."TO_zu_GP02.QM46");
END_REGION

REGION Network 10 (SCL): CL0x
   "Ventilstatus_einfach"(A_Ventil:= "A_CL01.QM51",
                          "Farbe HMI" => "Panel".Ventil."CL01.QM51");

   "Ventilstatus_einfach"(A_Ventil := "A_CL02.QM52",
                          "Farbe HMI" => "Panel".Ventil."CL02.QM52");
END_REGION
END_FUNCTION_BLOCK
